// TIA Portal V20 export
DATA_BLOCK "CallEquipment_DB"   // DB38
{ DB_Accessible_From_OPC_UA := 'FALSE' }
// stored: AssignedProDiagFB Unit1.Em6.ProDiag, DBAccessibleFromOPCUA false, DBAccessibleFromWebserver false, InstanceOfName Unit1.Em6.CallEquipment, InstanceOfType FB, Namespace Unit1.Em6
"Unit1.Em6.CallEquipment"
   // VAR_INPUT
   //    ZoneOperationEnable { ExternalWritable := 'False'} : "LWONIK_typeSafetyZoneManualOperation";
   // END_VAR
   // VAR_IN_OUT
   //    unitStatus : "LAF_typeUnitStatus";
   //    emFeedback : "LUC_typeEmFeedback";
   //    unitAlarmDB : "LAF_typeAlarms";
   // END_VAR
   // VAR
   //    InstHotPressLeftSequence { ExternalWritable := 'False'} : "Unit1.Em6.Sequence_1_HotPressLeft";
   //    instHotPressLeftHomeJob1 { ExternalWritable := 'False'} : "LAF_SelectJob";
   //    instHotPressLeftLoadJob2 { ExternalWritable := 'False'} : "LAF_SelectJob";
   //    instHotPressLeftInspectionJob3 { ExternalWritable := 'False'} : "LAF_SelectJob";
   //    instHotPressLeftUnloadJob4 { ExternalWritable := 'False'} : "LAF_SelectJob";
   //    instCmHotPressLeftSafetyPin { ExternalWritable := 'False'} : "LBC_DigitalSignalCn";
   //    instCmHotPressLeftJRDetect { ExternalWritable := 'False'} : "LBC_DigitalSignalCn";
   //    instCmHotPressLeftStageLiftFrontUpDown { ExternalWritable := 'False'} : "LBC_TwoWayActuatorCn";
   //    instCmHotPressLeftStageLiftRearUpDown { ExternalWritable := 'False'} : "LBC_TwoWayActuatorCn";
   //    instCmHotPressLeftStageLiftAllUpDown { ExternalWritable := 'False'} : "LBC_TwoWayActuatorCn";
   //    instCmHotPressLeftTemperature { ExternalWritable := 'False'} : "LER_Heater";
   //    instCmHotPressLeftServoPress { ExternalWritable := 'False'} : "LER_ServoPress";
   //    instCmHotPressLeftHistroy { ExternalWritable := 'False'} : "LER_ServoPressHistory";
   //    instManageAlarms { ExternalWritable := 'False'} : "LAF_ManageAlarms";
   //    instEventsPFE { ExternalWritable := 'False'} : "Unit1.Em6.EventsPFE";
   //    statUnitStatus { ExternalWritable := 'False'} : "LAF_typeUnitStatus";
   // END_VAR
   // VAR RETAIN
   //    statPartData { ExternalWritable := 'False'} : "LER_typePartData";
   // END_VAR
   // VAR
   //    statDataDelete { ExternalWritable := 'False'} : "LER_typePartData";
   //    statHistoryDeleteData { ExternalWritable := 'False'} : "LER_typeServoPressHistory";
   //    statClock { ExternalWritable := 'False'} : "LAF_typeGlobalClockMem";
   //    statTonTime { ExternalWritable := 'False'} : Array[0..999] of TON_TIME;
   //    statTofTime { ExternalWritable := 'False'} : Array[0..9] of TOF_TIME;
   //    statPulse { ExternalWritable := 'False'} : Array[0..999] of Bool;
   //    statNomalMode { ExternalWritable := 'False'} : Bool;
   //    statEnableManualCmds { ExternalWritable := 'False'} : Bool;
   //    statDoorOpenTemperature { ExternalWritable := 'False'} : "Safety.typeHotPressTempOk";
   //    statRunTemperature { ExternalWritable := 'False'} : Bool;
   //    "*** Interlock TwoWay ***" { S7_SetPoint := 'True'} : "LER_Axis_Homing";
   //    instCmHotPressLeftStageLiftFrontUpDownInterlock { S7_SetPoint := 'True'} : Array[0..2] of "LER_Actuator";
   //    instCmHotPressLeftStageLiftRearUpDownInterlock { S7_SetPoint := 'True'} : Array[0..2] of "LER_Actuator";
   //    instCmHotPressLeftStageLiftAllUpDownInterlock { S7_SetPoint := 'True'} : Array[0..2] of "LER_Actuator";
   //    HotPressLeftStageLiftFrontUpDown_Inpos : Array[0..2] of Struct
   //       "Int" : Array[1..10] of Bool;
   //    END_STRUCT;
   //    HotPressLeftStageLiftRearUpDown_Inpos : Array[0..2] of Struct
   //       "Int" : Array[1..10] of Bool;
   //    END_STRUCT;
   //    HotPressLeftStageLiftAllUpDown_Inpos : Array[0..2] of Struct
   //       "Int" : Array[1..10] of Bool;
   //    END_STRUCT;
   //    citi_Ptrig : Array[0..20] of Bool;
   //    citiTon : Array[0..20] of TON_TIME;
   //    citi : Time;
   //    citiTest : Array[0..20] of Bool;
   //    statReal : Array[0..9] of Real;
   //    instPFERecipe { S7_SetPoint := 'True'} : "Unit1.Em6.EventsPFE_Recipe";
   // END_VAR
BEGIN
END_DATA_BLOCK
